SUBAPPLICATION ACTION_SERVER_CANCEL_GOAL
  (* Standard: 61499-2 *)
  (* Version 1.0, 2023-04-02, Tim Hesse *)
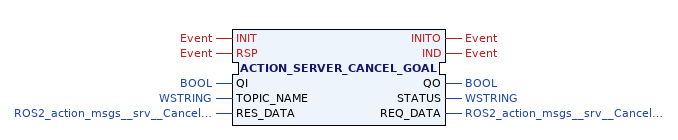
  EVENT_INPUT
    INIT; (* Initialization Request *)
    RSP;
  END_EVENT
  EVENT_OUTPUT
    INITO; (* Initialization Confirm *)
    IND;
  END_EVENT
  VAR_INPUT
    QI : BOOL; (* Input event qualifier *)
    TOPIC_NAME : WSTRING;
    RES_DATA : ROS2_action_msgs__srv__CancelGoal__Response;
  END_VAR
  VAR_OUTPUT
    QO : BOOL; (* Output event qualifier *)
    STATUS : WSTRING;
    REQ_DATA : ROS2_action_msgs__srv__CancelGoal__Request;
  END_VAR
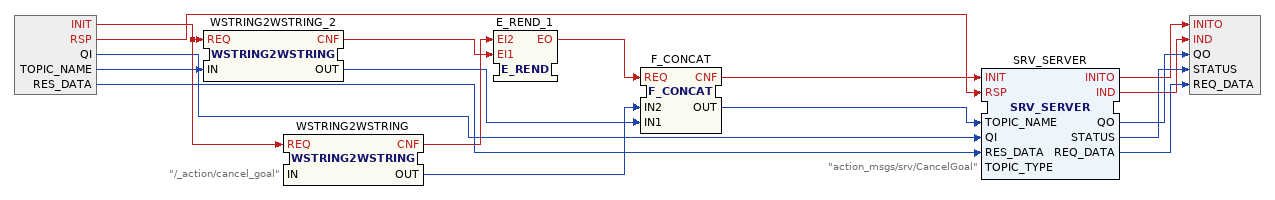
  FBS
    E_REND_1 : E_REND;
    WSTRING2WSTRING_2 : WSTRING2WSTRING;
    F_CONCAT : F_CONCAT;
    WSTRING2WSTRING : WSTRING2WSTRING(IN := "/_action/cancel_goal");
  END_FBS
  SUBAPPS
    SRV_SERVER : SRV_SERVER(TOPIC_TYPE := "action_msgs/srv/CancelGoal");
  END_SUBAPPS
  EVENT_CONNECTIONS
    E_REND_1.EO TO F_CONCAT.REQ;
    WSTRING2WSTRING.CNF TO E_REND_1.EI2;
    WSTRING2WSTRING_2.CNF TO E_REND_1.EI1;
    F_CONCAT.CNF TO SRV_SERVER.INIT;
    INIT TO WSTRING2WSTRING_2.REQ;
    INIT TO WSTRING2WSTRING.REQ;
    RSP TO SRV_SERVER.RSP;
    SRV_SERVER.INITO TO INITO;
    SRV_SERVER.IND TO IND;
  END_CONNECTIONS
  DATA_CONNECTIONS
    WSTRING2WSTRING.OUT TO F_CONCAT.IN2;
    WSTRING2WSTRING_2.OUT TO F_CONCAT.IN1;
    F_CONCAT.OUT TO SRV_SERVER.TOPIC_NAME;
    QI TO SRV_SERVER.QI;
    TOPIC_NAME TO WSTRING2WSTRING_2.IN;
    RES_DATA TO SRV_SERVER.RES_DATA;
    SRV_SERVER.QO TO QO;
    SRV_SERVER.STATUS TO STATUS;
    SRV_SERVER.REQ_DATA TO REQ_DATA;
  END_CONNECTIONS
END_SUBAPPLICATION
